FUNCTION_BLOCK TGenericCollection
VAR
   name : STRING;
END_VAR

//WIP. Consider making it runtime capable of change.

METHOD FB_init : BOOL
VAR_INPUT
   bInitRetains : BOOL; // if TRUE, the retain variables are initialized (warm start / cold start)
   bInCopyCode : BOOL; // if TRUE, the instance afterwards gets moved into the copy code (online change)
   T : Tc2_Utilities.T_Arg // provide type of the collection.
END_VAR
IF T.cbLen > 0 THEN

ELSE
   F_LogError();
END_IF
END_METHOD

END_FUNCTION_BLOCK

(* stored: Version 1.1.0.1, ProductVersion 3.1.4024.9
   POU TGenericCollection: Id {e481bb3a-f53c-455a-8869-ffee33fe2ff9}, SpecialFunc None
   Method FB_init: Id {a5a18c66-e929-46f3-b815-8b6ba56d0b05} *)
